(* CODESYS project statemachine_1022.library
   Author: Filippo Boido
   Placeholder: StateMachineLib
   Title: StateMachineLib
   Version: 1.0.2.2
   Company: FactoryAutomation

Project tree, tasks and I/O mapping:
  libraries: Tc2_Standard, * (Beckhoff Automation GmbH); Tc2_System, * (Beckhoff Automation GmbH); Tc3_Module, * (Beckhoff Automation GmbH); VersionLib, * (FactoryAutomation)
  DUTs/
    data type E_StateMachine
    data type E_TestUnitBusyStep
    data type ST_StateMachine
  GVLs/
  POUs/
    program MAIN [ST]
    function block StateMachine [ST]: ChangeState, Boot, Done, EndWait, Execute, Fault, Reset, Start, Wait, Busy, Error, Idle, Init, Prepare, Ready, Waiting
    function block TestFB [ST]: Busy, Error, Idle, Init, Prepare, Ready, Waiting
  VISUs/
  program Version [ST]
*)

// DUTs/E_StateMachine
{attribute 'to_string'}
TYPE E_StateMachine :
(
	eNoState := 0,
	eInit, 		
    eReady,
	ePrepare, 		
    eBusy, 		
    eWaiting, 	
    eIdle, 		
    eError 		
);
END_TYPE


(*	

				                   V  Boot()						
								   |  									 
                                   |
								<Init>
								   |
								   |	
                                   |  Start()
                                   |
                                   |
								<Ready> -----------<--------------+-------------<-----------+
								   |                              |                         |
                                   |                              |                         |
                                   |  Execute()                   |                         |
 								   | 							  |							|
                                   |                              |                         |
                                   |                              |   Reset()              |
 							   <Prepare>                          |                         |
 								   |                              |                         |
                                   |                              |                         |
                                   |                              |                         |
                   Wait()          |           Fault()            |                         |
	 <Waiting> ---<-------->--- <Busy> ----------->----------- <Error>                      |
				  EndWait() 	   |                                                        |
								   |	                                                    |
                                   |                                                 		|
                                   |                                                        |
								   |  Done()												|
								   |                                                        |
								   |                                                        |
								   |                                                        |
								<Idle> ---------------------->------------------------------+
								   
								   
Das erste Mal wo der FB aufgerufen wird, wird bBoot auf TRUE gesetzt und bleibt TRUE bis zum Neustart der Runtime.
Das heißt Init() wird selbstständig vom FB im ersten Zyklus aufgerufen.
Sobald Start() aufgerufen wird, wird Ready() ausgeführt, jedoch nur wenn die StateMachine sich im Init befindet.
Wenn Ready() läuft, kann Init() nicht mehr aufgerufen werden.
Durch Execute() wird der Zustand für ein Zyklus zu Prepare und anschließend zu Busy gewechselt.
Von hier aus wird entweder durch einen Fehler in den Error oder durch ein Wait() in den Waiting Zustand gewechselt.
Waiting kann nur zurück ins Busy und vom Error aus gehts nur nach Ready zurück.
Wenn Busy fertig ist wird für ein Zyklus Idle und dann wieder Ready aufgerufen.
							   
*)

// DUTs/E_TestUnitBusyStep
{attribute 'to_string'}
TYPE E_TestUnitBusyStep :
(
	eNO_STEP := 0,
	eWAITING_FOR_MATERIAL := 100
);
END_TYPE

// DUTs/ST_StateMachine
TYPE ST_StateMachine :
STRUCT
	uiInit 		: UINT;
	uiReady 	: UINT;
	uiBusy 		: UINT;
	uiWaiting 	: UINT;
	uiIdle 		: UINT;
	uiError 	: UINT;
END_STRUCT
END_TYPE

// POUs/MAIN
PROGRAM MAIN
VAR
	fbTest : TestFB;
END_VAR

fbTest();
fbTest.Execute();

END_PROGRAM

// POUs/TestFB
FUNCTION_BLOCK TestFB EXTENDS StateMachine 
VAR_INPUT
END_VAR
VAR_OUTPUT
	eTestUnitBusyStep : E_TestUnitBusyStep;
END_VAR
VAR
END_VAR

SUPER^();
eTestUnitBusyStep := stStateMachine.uiBusy;
Start();

METHOD PROTECTED Busy : BOOL
stStateMachine.uiBusy := eWAITING_FOR_MATERIAL;
END_METHOD

METHOD PROTECTED Error : BOOL
END_METHOD

METHOD PROTECTED Idle : BOOL
END_METHOD

METHOD PROTECTED Init : BOOL
END_METHOD

METHOD PROTECTED Prepare : BOOL
END_METHOD

METHOD PROTECTED Ready : BOOL
END_METHOD

METHOD PROTECTED Waiting : BOOL
END_METHOD

END_FUNCTION_BLOCK

// POUs/StateMachine
FUNCTION_BLOCK ABSTRACT StateMachine 
VAR_INPUT
END_VAR
VAR_OUTPUT
	sStateMachine : STRING;
END_VAR
VAR
	
	eStateMachine : E_StateMachine;
	stStateMachine : ST_StateMachine;
	bFirstCycle : BOOL := TRUE;
END_VAR

//sStateMachine := TO_STRING(eStateMachine);

Boot();

CASE eStateMachine OF

	eInit:
		Init();
	eReady:
		Ready();
	ePrepare:
		Prepare();
		eStateMachine := eBusy;
	eBusy:
		Busy();
	eIdle:
		Idle();
		eStateMachine := eReady;
	eWaiting:
		Waiting();
	eError:
		Error();
		
END_CASE

METHOD PRIVATE ChangeState : BOOL
VAR_INPUT
	eStateMachine : E_StateMachine;
END_VAR
THIS^.eStateMachine := eStateMachine;
END_METHOD

METHOD PROTECTED Boot : BOOL
VAR_INPUT
END_VAR
IF bFirstCycle
THEN
	ChangeState(eInit);
	bFirstCycle := FALSE;	
	Boot := TRUE;
END_IF
END_METHOD

METHOD PROTECTED Done : BOOL
VAR_INPUT
END_VAR
IF eStateMachine = eBusy
THEN
	ChangeState(eIdle);
	Done := TRUE;
END_IF
END_METHOD

METHOD PUBLIC EndWait : BOOL
VAR_INPUT
END_VAR
IF eStateMachine = eWaiting
THEN
	ChangeState(eBusy);
	EndWait := TRUE;
END_IF
END_METHOD

METHOD PUBLIC Execute : BOOL
VAR_INPUT
END_VAR
IF eStateMachine = eReady 
THEN
	ChangeState(ePrepare);
	Execute := TRUE;
END_IF
END_METHOD

METHOD PROTECTED Fault : BOOL
VAR_INPUT
END_VAR
IF eStateMachine = eBusy 
THEN
	ChangeState(eError);
	Fault := TRUE;
END_IF
END_METHOD

METHOD PUBLIC Reset : BOOL
VAR_INPUT
END_VAR
IF eStateMachine = eError 
THEN
	ChangeState(eReady);
	Reset := TRUE;
END_IF
END_METHOD

METHOD PROTECTED Start : BOOL
VAR_INPUT
END_VAR
IF eStateMachine = eInit 
THEN
	ChangeState(eReady);
	Start := TRUE;
END_IF
END_METHOD

METHOD PUBLIC Wait : BOOL
VAR_INPUT
END_VAR
IF eStateMachine = eBusy
THEN
	ChangeState(eWaiting);
	Wait := TRUE;
END_IF
END_METHOD

METHOD PROTECTED ABSTRACT  Busy : BOOL
VAR_INPUT
END_VAR
END_METHOD

METHOD PROTECTED ABSTRACT Error : BOOL
VAR_INPUT
END_VAR
END_METHOD

METHOD PROTECTED ABSTRACT Idle : BOOL
VAR_INPUT
END_VAR
END_METHOD

METHOD PROTECTED ABSTRACT Init : BOOL
VAR_INPUT
END_VAR
END_METHOD

METHOD PROTECTED ABSTRACT Prepare : BOOL
VAR_INPUT
END_VAR
END_METHOD

METHOD PROTECTED ABSTRACT Ready : BOOL
VAR_INPUT
END_VAR
END_METHOD

METHOD PROTECTED ABSTRACT Waiting : BOOL
VAR_INPUT
END_VAR
END_METHOD

END_FUNCTION_BLOCK

// Version
PROGRAM Version
VAR
END_VAR

(*
1.0.1.1:	Boido	010120

Added VersionLib and Verstion.txt to the project.

1.0.2.2:	Boido	020120

Version.txt replaced with Version PRG

*)

END_PROGRAM
